// TIA Portal project "hmi_13.11.23" (V16)

(* hardware
DEVICE "S71500/ET200MP station_1"  S7-1500 station
   slot 0: "Rail_0"  Rack  6ES7 590-1***0-0AA0
   slot 1: "PLC_1"  CPU 1512C-1 PN  6ES7 512-1CK01-0AB0  V2.8
      slot 3: "CPU display_1"  6ES7591-1AA00-0AA0
      slot 32768: "PROFINET interface_1"  X1
         slot 32769: "Port_1"  X1 P1
         slot 32770: "Port_2"  X1 P2
      slot 34817: "Virtual CP interface port_1"  Virtual CP interface port  Virtual CP interface port
DEVICE "HMI_1"  TP700 Comfort
   slot 0: "HMI_1"  TP700 Comfort  6AV2 124-0GC01-0AX0  16.0.0.0
   slot 1: "HMI_RT_1"  TP700 Comfort  6AV2 124-0GC01-0AX0  16.0.0.0
   slot 5: "HMI_1.IE_CP_1"  PROFINET Interface  16.0.0.0
      slot 1: "PROFINET Interface_1"  PROFINET Interface
         slot 1: "Port_1"  Port
         slot 2: "Port_2"  Port
   slot 7: "HMI_1.MPI/DP_CP_1"  MPI/DP Interface  16.0.0.0
*)

// ===== PLC "PLC_1"  CPU 1512C-1 PN =====

VAR_GLOBAL   // PLC tag table "Default tag table"
   "Clock_Byte" AT %MB1000 : Byte;
   "Clock_10Hz" AT %M1000.0 : Bool;
   "Clock_5Hz" AT %M1000.1 : Bool;
   "Clock_2.5Hz" AT %M1000.2 : Bool;
   "Clock_2Hz" AT %M1000.3 : Bool;
   "Clock_1.25Hz" AT %M1000.4 : Bool;
   "Clock_1Hz" AT %M1000.5 : Bool;
   "Clock_0.625Hz" AT %M1000.6 : Bool;
   "Clock_0.5Hz" AT %M1000.7 : Bool;
   "Start" AT %M1001.0 : Bool;
   "Reset" AT %M1001.1 : Bool;
   "Stop" AT %M1001.2 : Bool;
   "l_start" AT %M1001.3 : Bool;
   "l_reset" AT %M1001.4 : Bool;
   "Man" AT %M1001.5 : Bool;
   "l_Q1" AT %M1001.6 : Bool;
   "l_Q2" AT %M1001.7 : Bool;
END_VAR

ORGANIZATION_BLOCK "Main"   // OB1, LAD, ProgramCycle
TITLE = "Main Program Sweep (Cycle)"
{ S7_Optimized_Access := 'TRUE' }
VERSION : 0.1
   VAR_INPUT
      Initial_Call : Bool;   // Initial call of this OB
      Remanence : Bool;   // =True, if remanent data are available
   END_VAR
BEGIN
END_ORGANIZATION_BLOCK

(* ===== HMI "HMI_RT_1" =====
system functions are stored by id; their names below are inferred from use
connection "HMI_Connection_1": ETHERNET, S7_1500_OMS

HMI tags "Default tag table"
   "Start" : Bool = PLC Start AT %M1001.0, 100 ms
   "Reset" : Bool = PLC Reset AT %M1001.1, 100 ms
   "Stop" : Bool = PLC Stop AT %M1001.2, 100 ms
   "l_start" : Bool = PLC l_start AT %M1001.3, 100 ms
   "l_reset" : Bool = PLC l_reset AT %M1001.4, 100 ms
   "Man" : Bool = PLC Man AT %M1001.5, 100 ms
   "l_Q1" : Bool = PLC l_Q1 AT %M1001.6, 100 ms
   "l_Q2" : Bool = PLC l_Q2 AT %M1001.7, 100 ms

screen "Main screen" 800x480, template "Template_1"
   Button "Button_1" at 40,31 size 96x62; TextOff 'START'
      on Press: SetBit("Start")
      on Release: ResetBit("Start")
   Button "Button_2" at 246,31 size 96x62; TextOff 'STOP'
      on Release: ResetBit("Stop")
      on Press: SetBit("Stop")
   Button "Button_3" at 40,150 size 96x62; TextOff 'RESET'
      on Release: ResetBit("Reset")
      on Press: SetBit("Reset")
   Switch "Switch_1" at 254,132 size 148x88; CaptionText 'AUTO (0) MAN (1)'; TextOff 'OFF'; TextOn 'ON'
      ProcessValue <- "Man"
   SymbolLibrary "Symbol library_1" at 142,38 size 46x44
      Appearance <- "l_start"
   SymbolLibrary "Symbol library_2" at 142,161 size 46x44
      Appearance <- "l_reset"
   SymbolLibrary "Symbol library_3" at 12,255 size 65x61
      Appearance <- "l_Q1"
   SymbolLibrary "Symbol library_4" at 124,283 size 65x61
      Appearance <- "l_Q2"
   TextField "Text field_1" at 24,369 size 61x58; Text 'Q1'
   TextField "Text field_2" at 123,403 size 61x58; Text 'Q2'
*)